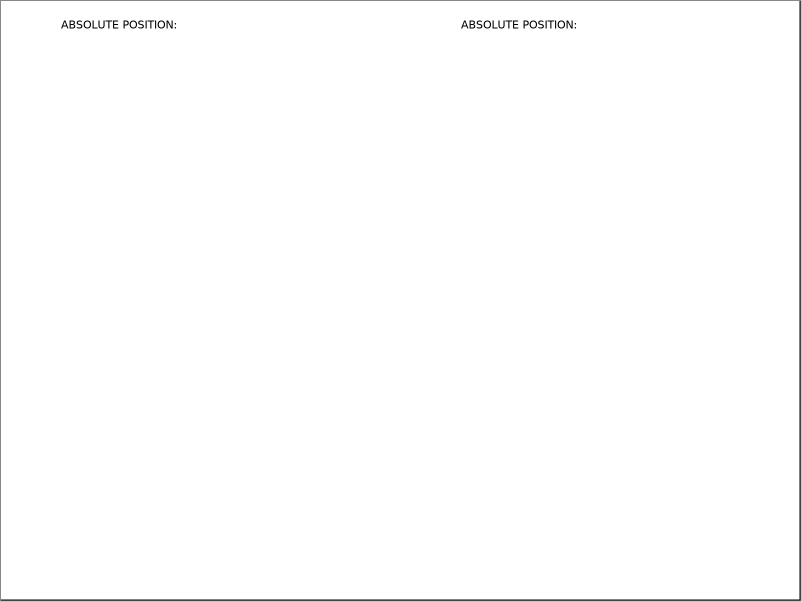
VISUALIZATION F24_Home  // 802x602
    Rectangle (0,0 800x600)
    Label (10,10 170x30), "ABSOLUTE POSITION:"
    Label (410,10 170x30), "ABSOLUTE POSITION:"
END_VISUALIZATION

(* stored: Version 1.1.0.1, ProductVersion 3.1.4022.7
   Visu F24_Home: Id {70c26a95-bac3-4445-8f02-b2fb33e2f1c1} *)
